TYPE RobotPose :
STRUCT
	x, y, theta,e : LREAL;
END_STRUCT
END_TYPE

(* stored: Version 1.1.0.1, ProductVersion 3.1.4024.11
   DUT RobotPose: Id {8acee726-7633-4cd0-abd1-ae09009eb4c5} *)
